// TIA Portal V20 export
DATA_BLOCK "BK28"   // DB272
// stored: MemoryReserve 100
   VAR
      "X10-1.PUSHER ROLLER Z-AXIS LIMIT SENSOR(-)" : Bool := FALSE;
      "X10-2.PUSHER ROLLER Z-AXIS HOME SENSOR" : Bool := FALSE;
      "X12-1.PUSH ROLLER BACKWARD" : Bool := FALSE;
      "X12-2.PUSH ROLLER FORWARD" : Bool := FALSE;
      "X14-1.SPARE" : Bool := FALSE;
      "X14-2.SPARE" : Bool := FALSE;
      "X16-1.PUSHER ROLLER Z-AXIS LIMIT SENSOR(+)" : Bool := FALSE;
      "X16-2.SPARE" : Bool := FALSE;
   END_VAR
BEGIN
END_DATA_BLOCK
